# B&R Automation Studio project CoffeeMachine
Automation Studio 4.12.4.107 SP; 9232
; technology packages: mappView 5.22.1

## Configuration Config1

CPU X20CP0484, AutomationRuntime G4.93, Build 4.1.2, Vc V4.73.0

### Task classes (Cpu.sw)
```
Cyclic#1 (cycle 10000 us, tolerance 10000 us):
  Program <- Program.prg
```

### Hardware
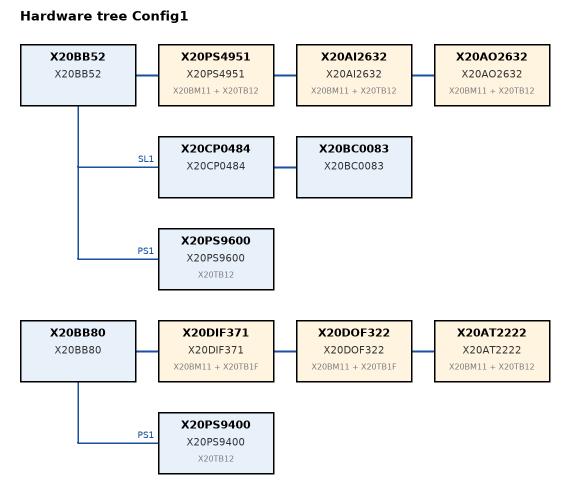
```
X20AI2632 : X20AI2632 v1.3.0.0  [SS1 -> X20TB12d.SS; SL -> X20BM11d.SL1]
  Supervision = off
X20AO2632 : X20AO2632 v1.2.0.0  [SS1 -> X20TB12e.SS; SL -> X20BM11e.SL1]
  Supervision = off
X20AT2222 : X20AT2222 v1.4.0.0  [SS1 -> X20TB12f.SS; SL -> X20BM11a.SL1]
  Supervision = off
X20BB52 : X20BB52 v1.2.0.0
  Connector IF6:
    CycleTime = 2000
X20BB80 : X20BB80 v1.1.0.0
X20BC0083 : X20BC0083 v2.14.0.0  [PLK1 -> X20CP0484.IF3 (NodeNumber=1) [Cable Type=PowerlinkCable, Length=10, Version=1.0.0.3]; SL -> X20BB80.SL1]
X20BM11 : X20BM11 v1.1.0.0  [X2X1 -> X20BB80.IF1]
X20BM11a : X20BM11 v1.1.0.0  [X2X1 -> X20BM11b.X2X2]
X20BM11b : X20BM11 v1.1.0.0  [X2X1 -> X20BM11.X2X2]
X20BM11c : X20BM11 v1.1.0.0  [X2X1 -> X20BB52.IF6]
X20BM11d : X20BM11 v1.1.0.0  [X2X1 -> X20BM11c.X2X2]
X20BM11e : X20BM11 v1.1.0.0  [X2X1 -> X20BM11d.X2X2]
X20CP0484 : X20CP0484 v1.6.0.0  [SL -> X20BB52.SL1]
  Connector IF2:
    ActivateDevice = 1
  ConfigurationID = CoffeeMachine_Config1
  Simulation = 1
  TimerDeviceType = SWIOTIMER
  Cyclic1Duration = 10000
  Cyclic1Tolerance = 10000
  Cyclic2Duration = 20000
  Cyclic2Tolerance = 20000
  Cyclic3Duration = 50000
  Cyclic3Tolerance = 50000
  Cyclic4Duration = 100000
  Cyclic4Tolerance = 100000
  Cyclic5Duration = 200000
  Cyclic5Tolerance = 200000
  Cyclic6Duration = 500000
  Cyclic6Tolerance = 500000
  Cyclic7Duration = 1000000
  Cyclic7Tolerance = 1000000
  Cyclic8Duration = 10000
  Cyclic8Tolerance = 30000000
  FileDevice1
  FileDeviceName1 = USER
  FileDevicePath1 = USER_PATH
  ActivateOpcUa = 1
  OpcUaInformationModels_PV_Version = 1
X20DIF371 : X20DIF371 v1.3.0.0  [SS1 -> X20TB1F.SS; SL -> X20BM11.SL1]
  Supervision = off
X20DOF322 : X20DOF322 v1.5.0.0  [SS1 -> X20TB1F1.SS; SL -> X20BM11b.SL1]
  Supervision = off
X20PS4951 : X20PS4951 v1.2.0.0  [SS1 -> X20TB12c.SS; SL -> X20BM11c.SL1]
  Supervision = off
X20PS9400 : X20PS9400 v1.8.0.0  [SS1 -> X20TB12b.SS; PS -> X20BB80.PS1]
X20PS9600 : X20PS9600 v1.6.0.0  [PS -> X20BB52.PS1; SS1 -> X20TB12.SS]
X20TB12 : X20TB12 v1.0.0.0
X20TB12b : X20TB12 v1.0.0.0
X20TB12c : X20TB12 v1.0.0.0
X20TB12d : X20TB12 v1.0.0.0
X20TB12e : X20TB12 v1.0.0.0
X20TB12f : X20TB12 v1.0.0.0
X20TB1F : X20TB1F v1.0.0.0
X20TB1F1 : X20TB1F v1.0.0.0
```

## Logical view

### Program Logical/Program

#### Types.typ
```iecst
TYPE
	COFFEE_enum :
		( (*Switch Case for coffee steps*)
		Wait,
		TimerRestart,
		CountMoney,
		Cancel,
		Dispense,
		Idle
		);
END_TYPE
```

#### Variables.var
```iecst
VAR
	COFFEESTEP : COFFEE_enum; (*Enum for coffee steps*)
	iVl_Flag : BOOL; (*Flag *)
	iMi_Cancel : BOOL; (*Cancel button*)
	iMi_COFFEE : BOOL; (*Coffee selection*)
	iMi_CoinFive : BOOL; (*5rs coin boolean to take hmi input*)
	iMi_CoinOne : BOOL; (*1rs coin boolean to take hmi input*)
	iMi_CoinTen : BOOL; (*10rs coin boolean to take hmi input*)
	iMi_CoinTwo : BOOL; (*2rs coin boolean to take hmi input *)
	iMi_COLDCOFFEE : BOOL; (*ColdCoffee selection*)
	iMi_COLDDRINK : BOOL; (*ColdDrink Selection*)
	iMi_DisTimeSet : {REDUND_UNREPLICABLE} INT := 5; (*Timer for dispense*)
	iMi_TEA : BOOL; (*Tea slection*)
	iMo_ChangeMoney : USINT; (*CHange money*)
END_VAR
VAR CONSTANT
	iMo_COFFEEPRICE : USINT := 10; (*price for coffee*)
	iMo_COLDCOFFEEPRICE : USINT := 15; (*price for coldcoffee*)
	iMo_COLDDRINKPRICE : USINT := 20; (*price for colddrink*)
END_VAR
VAR
	iMo_Display : STRING[80]; (*Display on hmi*)
END_VAR
VAR CONSTANT
	iMo_FIVE : USINT := 5; (*5rs coin*)
END_VAR
VAR
	iMo_GenDrink : STRING[80]; (*Generic drink*)
	iMo_GenPrice : USINT; (*generic price*)
	iMi_GoIntoCount : BOOL; (*process to count case*)
END_VAR
VAR CONSTANT
	iMo_ONE : USINT := 1; (*1rs coin*)
	iMo_TEAPRICE : USINT := 5; (*tea price*)
	iMo_TEN : USINT := 10; (*10rs coin*)
END_VAR
VAR
	iMo_TimerSmall : TON; (*Smalltimer for 10sec between two coins*)
END_VAR
VAR RETAIN
	iMo_TotalMoney : {REDUND_UNREPLICABLE} USINT; (*Totalmoeny inserted*)
END_VAR
VAR CONSTANT
	iMo_TWO : USINT := 2; (*2rs coin*)
END_VAR
VAR
	iVa_DispenseDrink : BOOL; (*Dispensing drink*)
	iVa_DisTimeSet : TON := (0); (*Timer for dispensing drink*)
	iVa_TimerFull : TON; (*40sec timer to put in all coins*)
	iVa_Svg : STRING[80]; (*Input string for svg to animate*)
	iVl_THIRTY : UDINT := 30; (*30 seconds for timer to diplay on hmi*)
END_VAR
VAR CONSTANT
	iVa_ONESEC : TIME := T#1s; (*1 second timer*)
END_VAR
VAR
	iVa_GoIntoIdle : BOOL; (*to go into idle case*)
	iMo_InsertCoin : UDINT; (*Insertcoin *)
	iVa_Cancel : TON; (*Cancel Button*)
	iVl_ChangeFlag : BOOL; (*Change buttton*)
	iVl_THIRTYTIMER : TIME := T#30S; (*Thirty second timer*)
	iVa_DisAnime : BOOL; (*Animation for Dispense*)
	iMo_Bar : UDINT; (*Bar value*)
	iMo_BarMax : INT; (*Bar max value*)
END_VAR
VAR RETAIN
	iMo_TotalInsertMoney : INT; (*Total money inserted till now*)
END_VAR
VAR
	iMo_PieCoffee : INT; (*Pie chart coffee counts*)
	iMo_PieTea : INT; (*Pie chart  tea counts*)
	iMo_PieCD : INT; (*Pie chart colddrink counts*)
	iMo_PieCC : INT; (*Pie chart colcounts*)
END_VAR
```

#### Main.st
```iecst
(*|ŻŻŻŻŻŻŻŻŻŻŻŻŻŻŻŻŻŻŻŻŻŻŻŻŻŻŻŻŻŻŻŻŻŻŻŻŻŻŻŻŻŻŻŻŻŻŻŻŻŻŻŻŻŻŻŻŻŻŻŻŻŻŻŻŻŻŻŻŻŻŻŻŻŻŻŻŻŻŻŻŻŻŻŻŻŻŻŻŻŻŻŻŻŻŻŻŻŻŻŻŻŻŻŻŻŻŻŻŻŻ|*)
(*| Copyright      :-  B&R Industrial Automation GmbH															 |*)
(*| Contact Person :-  maskeu																					 |*)
(*|——————————————————————————————————————————————————————————————————————————————————————————————————————————————|*)
(*| System       :- X20CP0484 																					 |*)
(*| Task Name    :-  Coffee Machine	                                                                	         |*)
(*| Auther Name  :-  maskeu																						 |*)
(*| Created Date :-  October 10, 2023 																		   	 |*)
(*| Task Class   :-  Task Class# Task Class No 1                                                                 |*)
(*| Task Time    :-  Task Timing 10mSec                                                                          |*)
(*| AS Version   :-  AS 4.12.4.107 SP                                                                            |*)
(*|——————————————————————————————————————————————————————————————————————————————————————————————————————————————|*)
(*| Description  :-  Coffee Machine			       	                                                             |*)
(*|______________________________________________________________________________________________________________|*)

PROGRAM _INIT
	//Full timer to put coins
	iVa_TimerFull.PT	:=T#40s;
	iMo_TimerSmall.PT	:=T#10s;
	// Cancel Time
	iVa_Cancel.PT		:=T#1s;
	iVa_Cancel.Q;
END_PROGRAM

PROGRAM _CYCLIC
	// ProgressBar max value
	iMo_BarMax			:=TIME_TO_INT(iVa_DisTimeSet.PT-iVa_ONESEC);
	//two seconds buffer time for dispensing
	iVa_DisTimeSet.PT	:=INT_TO_TIME(iMi_DisTimeSet * 1000)+iVa_ONESEC+iVa_ONESEC ;
	//if cancel is pressed cancel state
	IF iMi_Cancel = TRUE THEN
		COFFEESTEP 		:=Cancel;
	END_IF;

	//Enum for the coffeesteps
	CASE COFFEESTEP OF

		// Wait State waiting for user to give inputs
		Wait:
			IF iMo_TotalMoney>0 THEN
				iMo_ChangeMoney		:=iMo_TotalMoney;
				iMo_TotalMoney		:=0;
			ELSE
				iMo_TotalMoney		:=0;
			END_IF;
			IF iMi_GoIntoCount THEN
				iVa_TimerFull.IN	:=TRUE;
				iMo_TimerSmall.IN	:=TRUE;
				COFFEESTEP			:= CountMoney;
			END_IF;
			IF iVa_TimerFull.Q	=TRUE THEN
				COFFEESTEP		:=Idle;
			END_IF

			//If any drink is selected then it will become true and timer will start
			IF iMi_TEA=TRUE THEN
				iMo_GenDrink		:='TEA';
				iMo_GenPrice		:=iMo_TEAPRICE;
				iMi_TEA				:=FALSE;
				iVa_TimerFull.IN	:=TRUE;
			ELSIF iMi_COFFEE=TRUE THEN
				iMo_GenDrink		:= 'COFFEE';
				iMo_GenPrice		:=iMo_COFFEEPRICE;
				iMi_COFFEE			:=FALSE;
				iVa_TimerFull.IN	:=TRUE;
			ELSIF iMi_COLDDRINK=TRUE THEN
				iMo_GenDrink		:='COLDDRINK';
				iMo_GenPrice		:=iMo_COLDDRINKPRICE;
				iMi_COLDDRINK		:=FALSE;
				iVa_TimerFull.IN	:=TRUE;
			ELSIF iMi_COLDCOFFEE=TRUE THEN
				iMo_GenDrink		:='COLDCOFFEE';
				iMo_GenPrice 		:=iMo_COLDCOFFEEPRICE;
				iMi_COLDCOFFEE		:=FALSE;
				iVa_TimerFull.IN	:=TRUE;
			END_IF;

			// CountMoney State Money Inserted will be counted
		CountMoney:
			iVl_ChangeFlag			:=FALSE;
			iMi_GoIntoCount			:=FALSE;
			iMo_TimerSmall.IN		:=TRUE;

			// when timer ends it will go into idle state
			IF iVa_TimerFull.Q=TRUE OR iMo_TimerSmall.Q=TRUE THEN
				iVa_GoIntoIdle		:=TRUE;
				COFFEESTEP			:=Cancel;
			END_IF;

			//if timer of 10sec and 40sec collides then following block will execute
			IF iVa_TimerFull.ET<iVl_THIRTYTIMER THEN
				iMo_InsertCoin		:=iMo_TEN-TIME_TO_UDINT(iMo_TimerSmall.ET)/1000;
			ELSE
				iMo_InsertCoin		:=iVl_THIRTY+iMo_TEN-TIME_TO_UDINT(iVa_TimerFull.ET)/1000;
			END_IF;

			// when timer ends it will go into idle state
			IF iMo_TotalMoney>=iMo_GenPrice THEN
				iMo_Display			:='';
				iVa_DisTimeSet.IN	:=TRUE;
				COFFEESTEP			:=Dispense;
			ELSE
				iMo_Display:= 'Please Insert The Money';
			END_IF;

			//if any coin becomes true it will get added into total money
			IF iMi_CoinOne=TRUE THEN
				iMo_TotalMoney	:=iMo_TotalMoney + iMo_ONE;
				COFFEESTEP		:=TimerRestart;
			END_IF;
			IF iMi_CoinTwo = TRUE THEN
				iMo_TotalMoney	:=iMo_TotalMoney+iMo_TWO;
				COFFEESTEP		:=TimerRestart;
			END_IF;
			IF iMi_CoinFive=TRUE THEN
				iMo_TotalMoney 	:=iMo_TotalMoney+iMo_FIVE;
				COFFEESTEP		:=TimerRestart;
			END_IF;
			IF iMi_CoinTen=TRUE THEN
				iMo_TotalMoney 	:=iMo_TotalMoney+iMo_TEN;
				COFFEESTEP		:=TimerRestart;
			END_IF;

			// TimeRestart State TimerSmall will be restarted
		TimerRestart:
			iMo_TimerSmall.IN	:=FALSE;
			iMi_CoinFive		:=FALSE;
			iMi_CoinOne			:=FALSE;
			iMi_CoinTwo			:=FALSE ;
			iMi_CoinTen			:=FALSE;
			iVl_Flag			:=TRUE;
			COFFEESTEP			:=CountMoney;

			// Dispense State Drink will be out
			//concating strings to give svh animation
			//iVa_DisAnime- Is for animation of dispensing
		Dispense:
			iVa_DispenseDrink	:=TRUE;
			iMo_ChangeMoney		:=iMo_TotalMoney-iMo_GenPrice;
			iMo_Bar				:=TIME_TO_INT(iVa_DisTimeSet.ET);

			//paper svg animation code block
			IF iVa_DisTimeSet.ET<iVa_ONESEC THEN
				iVa_Svg			:='[{"select":"#cup","duration":1000,"translate":[190,0]}]';
				iMo_Display		:='Put the Cup';
				iVa_DisAnime	:=FALSE;
			ELSIF iVa_DisTimeSet.ET>iVa_DisTimeSet.PT - iVa_ONESEC THEN
				iVa_Svg			:='[{"select":"#cup","duration":1000,"translate":[0,0]}]';
				iMo_Display		:='Enjoy the Drink';
				iVa_DisAnime	:=FALSE;
				iMo_Bar			:=0;
			ELSE
				iMo_Display:='Dispensing the Drink';
				iVa_DisAnime:=TRUE;
			END_IF;
			IF iVa_DisTimeSet.Q = TRUE THEN
				COFFEESTEP		:=Idle;
			END_IF;

			//cancel button state
		Cancel:
			iMo_Bar					:=0;
			iMi_Cancel 				:=FALSE;
			iVa_Cancel.IN			:=TRUE;
			iVa_DisAnime			:=FALSE;
			iVa_Svg					:='[{"select":"#cup","translate":[0,0]}]';
			IF iVa_Cancel.Q=TRUE THEN
				COFFEESTEP			:=Idle;
			END_IF

			//if cancelled and money is inserted it will refund the moneuy
			IF iMo_TotalMoney>0 AND iVa_DispenseDrink=FALSE THEN
				iMo_TotalInsertMoney:=iMo_TotalInsertMoney+iMo_TotalMoney;
				iMo_ChangeMoney		:=iMo_TotalMoney;
				iMo_TotalMoney		:=0;
				iVl_ChangeFlag		:=TRUE;
			ELSE
				iMo_TotalMoney		:=0;
			END_IF;

			//Everything will be off in Idle state
		Idle:
			IF iMo_GenDrink = 'COFFEE'THEN
				iMo_PieCoffee:=iMo_PieCoffee+1;
			ELSIF iMo_GenDrink = 'TEA'THEN
				iMo_PieTea:=iMo_PieTea+1;
			ELSIF iMo_GenDrink = 'COLDCOFFEE'THEN
				iMo_PieCC:=iMo_PieCC+1;
			ELSIF iMo_GenDrink = 'COLDDRINK'THEN
				iMo_PieCD:=iMo_PieCD+1;
			END_IF;
			iMo_TotalInsertMoney	:=iMo_TotalInsertMoney+iMo_TotalMoney;
			iMo_Bar					:=0;
			iMo_TotalMoney			:=0;
			iVa_GoIntoIdle			:=FALSE;
			iMo_GenDrink			:='';
			iMo_GenPrice			:=0;
			iVa_DispenseDrink		:=FALSE;
			IF iVl_ChangeFlag=FALSE THEN
				iMo_ChangeMoney		:=0;
			END_IF;
			iMo_TotalMoney			:=0;
			iVa_TimerFull.IN		:=FALSE;
			iMo_TimerSmall.IN		:=FALSE;
			iVa_DisTimeSet.IN		:=FALSE;
			iVa_Cancel.IN			:=FALSE;
			iVa_DisAnime			:=FALSE;
			iMo_InsertCoin			:=0;
			iVa_Svg					:='[{"select":"#cup","translate":[0,0]}]';
			COFFEESTEP				:=Wait;
	END_CASE;
	//starting all timers
	iVa_TimerFull();
	iMo_TimerSmall();
	iVa_DisTimeSet();
	iVa_Cancel();
END_PROGRAM

PROGRAM _EXIT

END_PROGRAM
```
